// Gets the lower bound index of the array of specified type.
FUNCTION F_GetIntArrayLowerBound : T_Position // The lower bound index of the specified array.
VAR_IN_OUT
	arArray : ARRAY[*] OF INT; // The array to query.
END_VAR

F_GetIntArrayLowerBound := LOWER_BOUND(arArray, 1);

END_FUNCTION

(* stored: Version 1.1.0.1
   POU F_GetIntArrayLowerBound: Id {047c2235-5942-0980-3437-bd601a15fa21}, SpecialFunc None *)
